FUNCTION_BLOCK OR_2_BOOL (* FB to calculate boolean OR (generic FB) *)
  (* Standard: 61131-3; Classification: standard boolean function; Description: Copyright (c) 2014, 2024 Profactor GmbH, HR Agrartechnik GmbH This program and the accompanying materials are made available under the terms of the Eclipse Public License 2.0 which is available at https://www.eclipse.org/legal/epl-2.0/ SPDX-License-Identifier: EPL-2.0 *)
  (* Version 1.0, 2014-10-11, Matthias Plasch, Profactor GmbH *)
  (* Version 1.1, 2025-03-04, Franz Höpfinger, HR Agrartechnik GmbH, copy OR_2 and made OR_2_BOOL *)
  PACKAGE iec61131::booleanOperators;
  {SET_ATTRIBUTE(eclipse4diac::core::GenericClassName, 'GEN_OR_BOOL')}
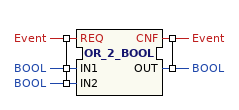
  EVENT_INPUT
    REQ WITH IN1, IN2; (* Normal Execution Request *)
  END_EVENT
  EVENT_OUTPUT
    CNF WITH OUT; (* Execution Confirmation *)
  END_EVENT
  VAR_INPUT
    IN1 : BOOL; (* OR input 1 *)
    IN2 : BOOL; (* OR input 2 *)
  END_VAR
  VAR_OUTPUT
    OUT : BOOL; (* OR result *)
  END_VAR
END_FUNCTION_BLOCK
